INTERFACE I_Enumerable EXTENDS __SYSTEM.IQueryInterface

METHOD PUBLIC GetEnumerator : I_ForwardEnumerator
END_METHOD

END_INTERFACE

(* stored: Version 1.1.0.1, ProductVersion 3.1.4024.12
   Itf I_Enumerable: Id {7db00eea-9f15-4284-ae07-5b26eba867a2}
   Method GetEnumerator: Id {aae136b0-94ef-4f19-bb74-e5527a3b8ee6} *)
